FUNCTION_BLOCK Room_State_SystemOff EXTENDS Room_State
VAR_INPUT
END_VAR
VAR_OUTPUT
END_VAR
VAR
END_VAR

METHOD CanDeactivate : BOOL
CanDeactivate := NOT _ctx.priv.bSysOff;
END_METHOD

METHOD OnEntry
_ctx.io.bOpenValves := FALSE;

_ctx.priv.bActive := FALSE;
_ctx.priv.bReady := FALSE;

_ctx.hmi.sStatusText := 'Central Heating is OFF';
_ctx.hmi.nStatusColor := COL.RED.Raw;

_ctx.hmi.bHideReset := FALSE;
END_METHOD

END_FUNCTION_BLOCK

(* stored: Version 1.1.0.1
   POU Room_State_SystemOff: Id {7c3aebcd-399b-4bac-9540-75fee170c6b7}, SpecialFunc None
   Method CanDeactivate: Id {8b2b34d2-b92c-4409-9ead-dd6ea6d63e93}
   Method OnEntry: Id {2165c4dc-33f4-4316-b0a7-0e9b5038a5aa} *)
